// TIA Portal V18 export
ORGANIZATION_BLOCK "PID Cyclic interrupt"   // OB30, FBD, CyclicInterrupt
{ S7_Optimized_Access := 'TRUE' }
VERSION : 0.1
// stored: AutoNumber true, IsIECCheckEnabled false, SetENOAutomatically false
   VAR_INPUT
      Initial_Call : Bool;   // Initial call of this OB
      Event_Count : Int;   // Events discarded
   END_VAR
BEGIN

REGION Network 1: Utility_PID
   // Utility_PID
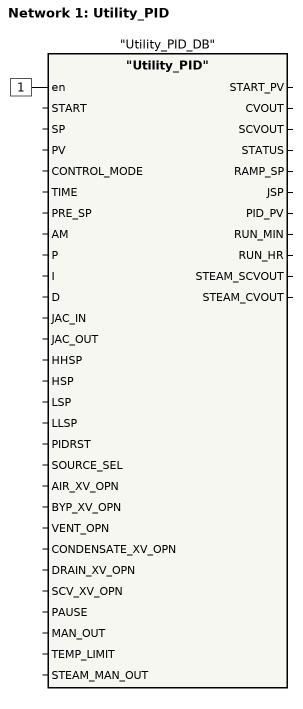
   IF 1 THEN
       "Utility_PID_DB"();   // "Utility_PID"
   END_IF;
END_REGION
END_ORGANIZATION_BLOCK
